// TIA Portal project "TestCase3_S1200_Zonder_Fouten" (V18)

(* hardware
DEVICE "S7-1200 station_1"  S7-1200 Station
   slot 0: "Rack_0"  S7-1200 Rack  Rack  V1.0
   slot 1: "PLC_1"  CPU 1212C DC/DC/DC  6ES7 212-1AE40-0XB0  V4.6
*)

// ===== PLC "PLC_1"  CPU 1212C DC/DC/DC =====

VAR_GLOBAL   // PLC tag table "Default tag table"
   "A" AT %I0.0 : Bool;
   "B" AT %I0.1 : Bool;
   "C" AT %I0.2 : Bool;
   "D" AT %I0.3 : Bool;
   "E" AT %I0.4 : Bool;
   "X" AT %Q0.0 : Bool;
END_VAR

DATA_BLOCK "Data_block_1_Inputs"   // DB1
{ S7_Optimized_Access := 'FALSE' }
VERSION : 0.1
   VAR
      "A" : Bool;
      "B" : Int;
      C : Int;
   END_VAR
BEGIN
END_DATA_BLOCK

DATA_BLOCK "Data_block_2_Outputs"   // DB2
{ S7_Optimized_Access := 'FALSE' }
VERSION : 0.1
   VAR
      "A" : Byte;
      "B" : Word;
      C : DWord;
      D : Int;
      "E" : DInt;
      F : Real;
   END_VAR
BEGIN
END_DATA_BLOCK

ORGANIZATION_BLOCK "Main"   // OB1, FBD, ProgramCycle
TITLE = "Main Program Sweep (Cycle)"
{ S7_Optimized_Access := 'TRUE' }
VERSION : 0.1
   VAR_INPUT
      Initial_Call : Bool;   // Initial call of this OB
      Remanence : Bool;   // =True, if remanent data are available
   END_VAR
   VAR_TEMP   // added for the SCL form of the ladder/FBD networks
      _w1 : Bool;
   END_VAR
BEGIN

REGION Network 1
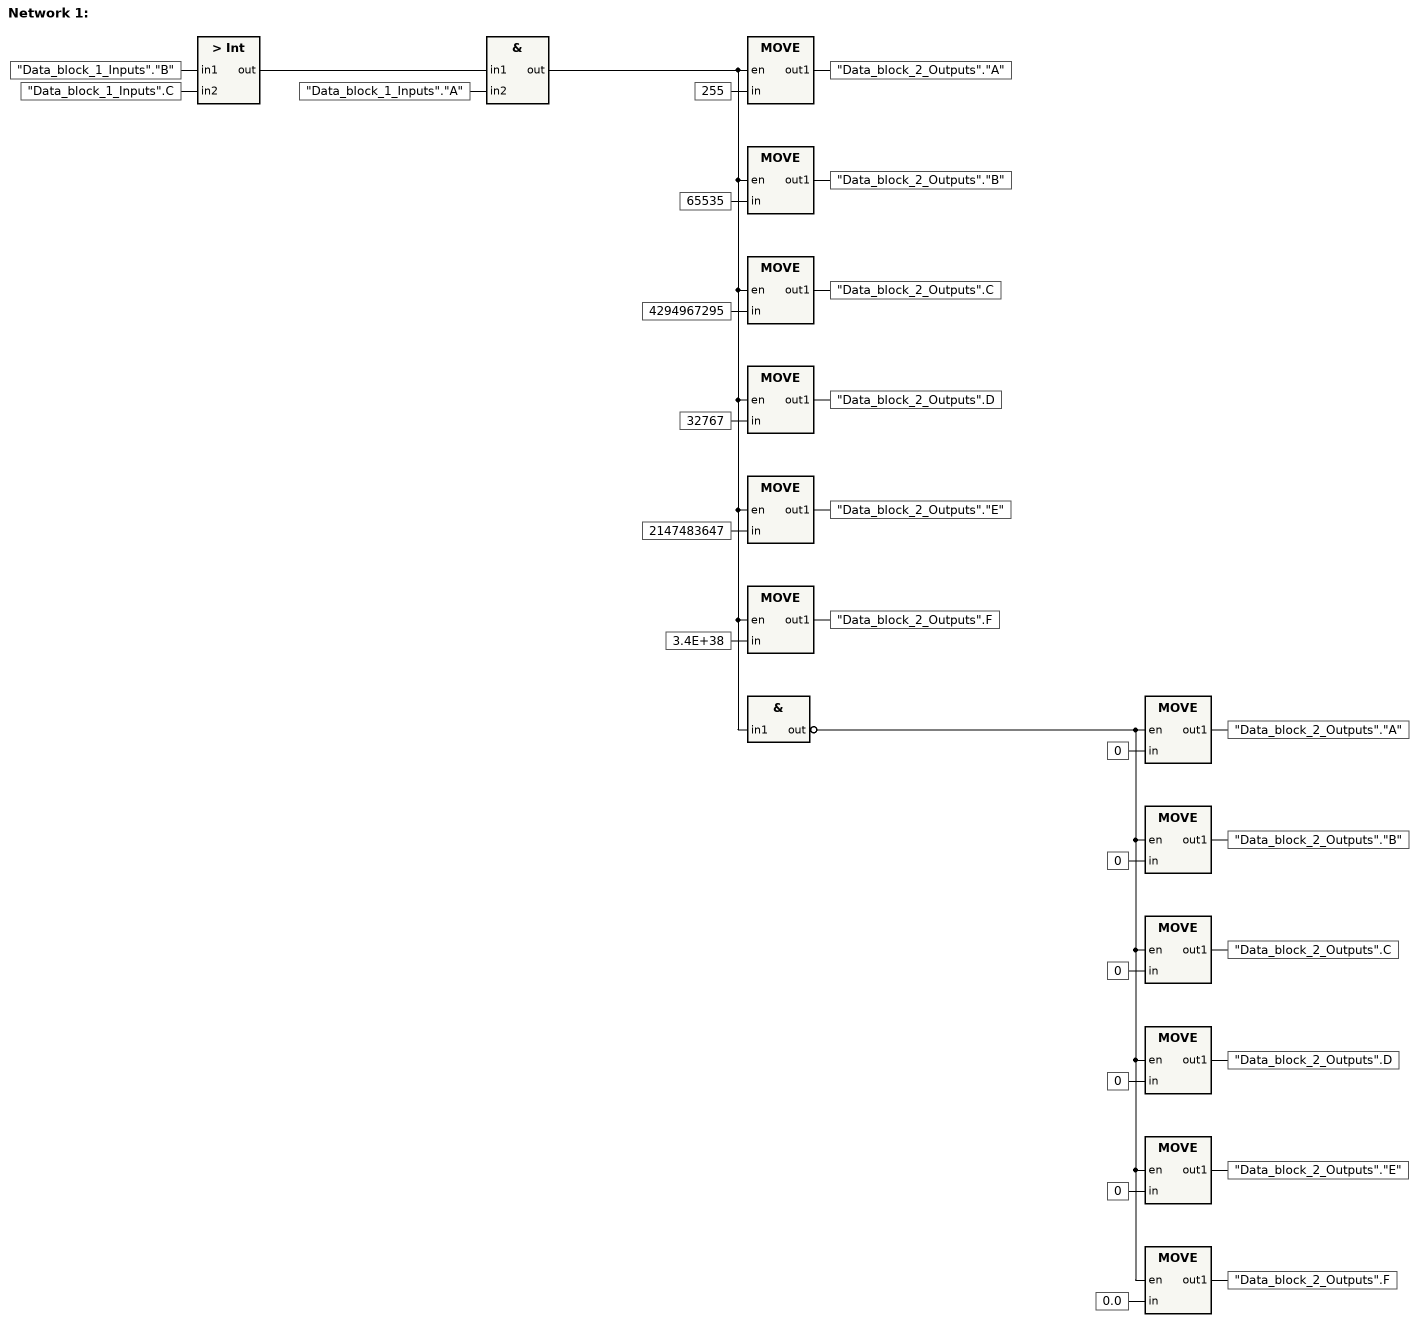
   #_w1 := ("Data_block_1_Inputs"."B" > "Data_block_1_Inputs".C) AND "Data_block_1_Inputs"."A";
   IF #_w1 THEN
       "Data_block_2_Outputs"."A" := 255;
       "Data_block_2_Outputs"."B" := 65535;
       "Data_block_2_Outputs".C := 4294967295;
       "Data_block_2_Outputs".D := 32767;
       "Data_block_2_Outputs"."E" := 2147483647;
       "Data_block_2_Outputs".F := 3.4E+38;
   END_IF;
   IF NOT #_w1 THEN
       "Data_block_2_Outputs"."A" := 0;
       "Data_block_2_Outputs"."B" := 0;
       "Data_block_2_Outputs".C := 0;
       "Data_block_2_Outputs".D := 0;
       "Data_block_2_Outputs"."E" := 0;
       "Data_block_2_Outputs".F := 0.0;
   END_IF;
END_REGION
END_ORGANIZATION_BLOCK